FUNCTION_BLOCK fbConveyorCtrl
VAR_INPUT
	bEnable		: BOOL;
	bRapidPB	: BOOL;
	bZone1Sensor	: BOOL;
	bZone2Sensor	: BOOL;
	bEndZoneSensor	: BOOL;
	diZone1BasketConfirmDelayTime	: DINT;
	diZone2BasketConfirmDelayTime	: DINT;
	diEndZoneBasketConfirmDelayTime	: DINT;
	diRapidPBDelayTime	: DINT;

	bLdBasketZone1MemoryBit: BOOL;
	bEmergencyStop: BOOL;
END_VAR
VAR_OUTPUT
	bMotorOnOff	: BOOL;
END_VAR
VAR
	TON1: TON;
	TRIG1: R_TRIG;
	bMotorStopBit: BOOL;
	TON2: TON;
	Trig2: R_TRIG;
	TON3: TON;
	RampIn: BOOL;
	TON4: TON;
	bConvAutoCut: BOOL;
	CVDelayOff : BOOL;
	TON5: TON;
END_VAR

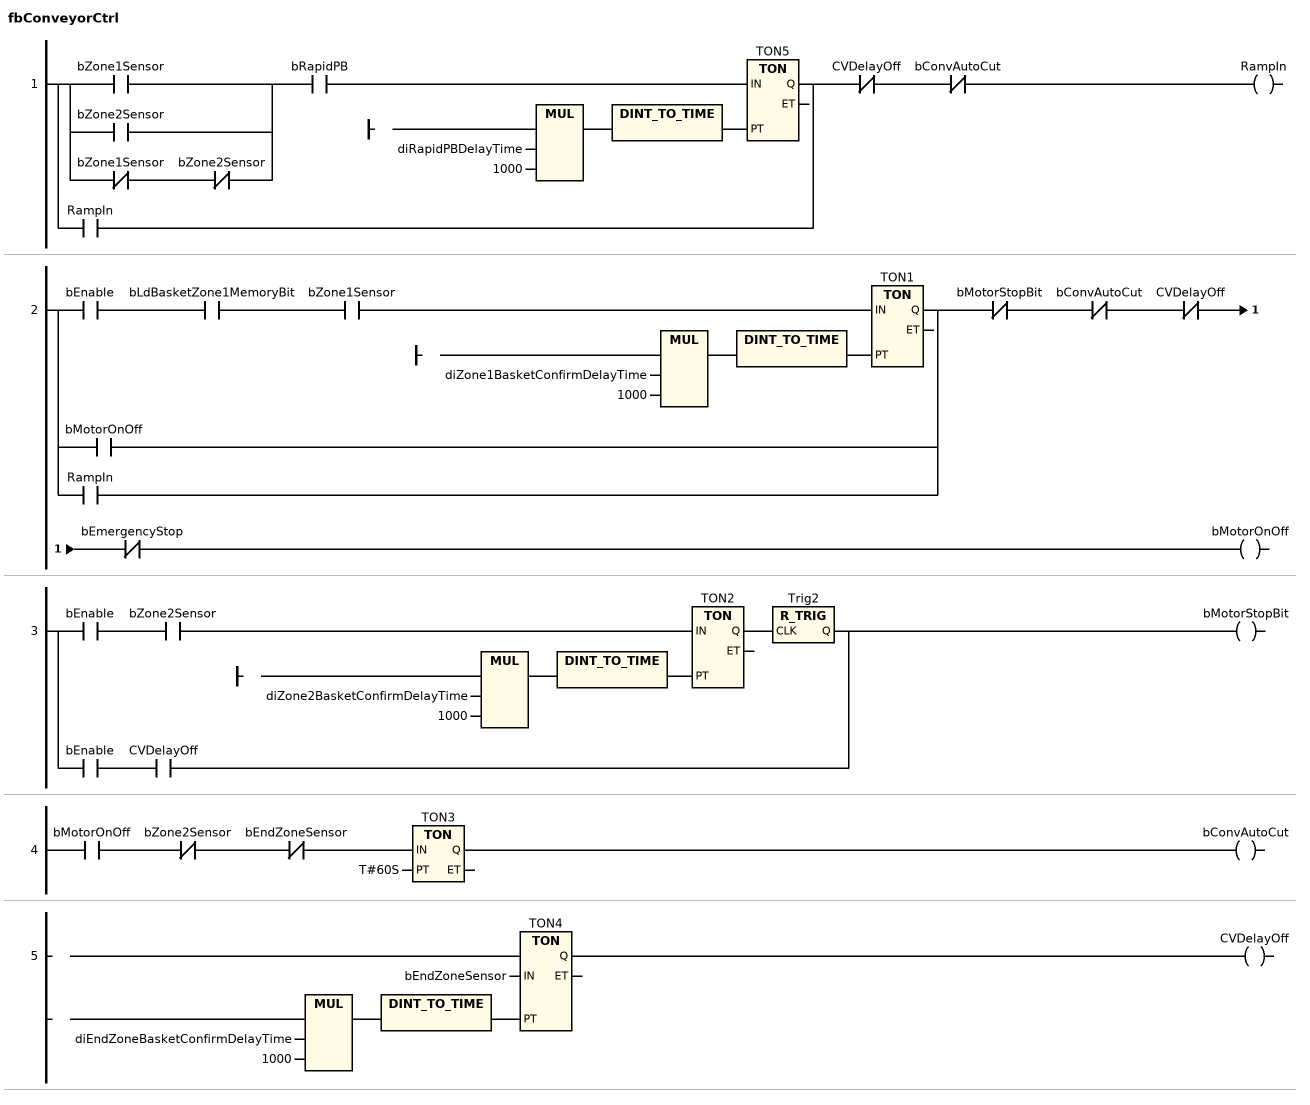
// NETWORK 1
TON5(IN := (bZone1Sensor OR bZone2Sensor OR NOT bZone1Sensor AND NOT bZone2Sensor) AND bRapidPB, PT := DINT_TO_TIME(diRapidPBDelayTime * 1000)); // TON
RampIn := (TON5.Q OR RampIn) AND NOT CVDelayOff AND NOT bConvAutoCut;

// NETWORK 2
TON1(IN := bEnable AND bLdBasketZone1MemoryBit AND bZone1Sensor, PT := DINT_TO_TIME(diZone1BasketConfirmDelayTime * 1000)); // TON
bMotorOnOff := (TON1.Q OR bMotorOnOff OR RampIn) AND NOT bMotorStopBit AND NOT bConvAutoCut AND NOT CVDelayOff AND NOT bEmergencyStop;

// NETWORK 3
TON2(IN := bEnable AND bZone2Sensor, PT := DINT_TO_TIME(diZone2BasketConfirmDelayTime * 1000)); // TON
Trig2(CLK := TON2.Q); // R_TRIG
bMotorStopBit := Trig2.Q OR bEnable AND CVDelayOff;

// NETWORK 4
TON3(IN := bMotorOnOff AND NOT bZone2Sensor AND NOT bEndZoneSensor, PT := T#60S); // TON
bConvAutoCut := TON3.Q;

// NETWORK 5
TON4(IN := bEndZoneSensor, PT := DINT_TO_TIME(diEndZoneBasketConfirmDelayTime * 1000)); // TON
CVDelayOff := TON4.Q;

END_FUNCTION_BLOCK

(* stored: Version 1.1.0.1, ProductVersion 3.1.4024.12
   POU fbConveyorCtrl: Id {1ec8b500-61d8-41d3-8de5-dff0525f8852}, SpecialFunc None *)
